// TIA Portal V20 export
DATA_BLOCK "T1-A ARUNC HMI"   // DB1202
{ S7_Optimized_Access := 'TRUE' }
AUTHOR : SAS
// stored: AutoNumber false, IsRetainMemResEnabled true, MemoryReserve 100, RetainMemoryReserve 100
   VAR
      Conditions : Struct
         CG : "Pop_Up_Aux";   // General conditions
         CA : "Pop_Up_Aux";   // Start Auto mode conditions
         SC : "Pop_Up_Aux";   // Start cycle conditions
         MOV_UP : "Pop_Up_Aux";   // Movement interlocks Up
      END_STRUCT;
      HMI : Struct
         PB : Struct
            s0 : Bool;
            s1 : Bool;
            s2 : Bool;
            s3 : Bool;
            s4 : Bool;
            Pause : Bool;   // Pause
            s6 : Bool;
            s7 : Bool;
            s8 : Bool;
            s9 : Bool;
            s10 : Bool;
            s11 : Bool;
            s12 : Bool;
            s13 : Bool;
            s14 : Bool;
            s15 : Bool;
         END_STRUCT;
         ST : Struct
            s0 : Bool;
            s1 : Bool;
            s2 : Bool;
            s3 : Bool;
            s4 : Bool;
            Pause : Bool;   // Pause
            s6 : Bool;
            s7 : Bool;
            s8 : Bool;
            s9 : Bool;
            "ST Machine" : Int;   // Device label status (0=EME, 1=Safe, 2=Fault, 3=Run, 4=Stopped)
            "ST Sequencer step" : Int;   // Sequencer step
         END_STRUCT;
      END_STRUCT;
   END_VAR
BEGIN
   // Conditions.CG.Conditions.n1 : Tensiune Alimentare OK
   // Conditions.CA.Conditions.n1 : Conditiie Generale
   // Conditions.CA.Conditions.n2 : Aruncator Jos
   // Conditions.SC.Conditions.n1 : Initial Conditions
   // Conditions.SC.Conditions.n2 : Piece Presence
   // Conditions.SC.Conditions.n3 : Tracking OK
   // Conditions.SC.Conditions.n4 : Condition of movement
   // Conditions.SC.Conditions.n5 : Sel. Incarca Cuptor calitor sin T1-A
   // Conditions.SC.Conditions.n6 : T1-A role Stop
   // Conditions.SC.Conditions.n7 : T1-A role Free
   // Conditions.SC.Conditions.n8 : Production Blocare
   // Conditions.SC.Conditions.n9 : Calire Consents
   // Conditions.MOV_UP.Conditions.n1 : Permanent Conditions
END_DATA_BLOCK
